// TIA Portal V15.1 export
// export: Created 2024-06-21T08:40:52.6402099Z, ExportSetting WithDefaults, DisplayName Totally Integrated Automation Portal, DisplayVersion V15.1 Update 5, DisplayName TIA Portal Openness, DisplayVersion V15.1 Update 5, DisplayName SINAMICS Startdrive Advanced, DisplayVersion V15.1, DisplayName G130, G150, S120, S150, SINAMICS MV, S210, DisplayVersion V15.1, DisplayName G110M, G120, G120C, G120D, G120P, DisplayVersion V15.1, DisplayName STEP 7 Professional, DisplayVersion V15.1 Update 5, DisplayName STEP 7 Safety, DisplayVersion V15.1, DisplayName WinCC Professional, DisplayVersion V15.1 Update 5, DisplayName SIMATIC Visualization Architect, DisplayVersion V15.1
FUNCTION_BLOCK "LHMIResetStart"   // FB1006, FBD
TITLE = LHMIResetStart
{ S7_Optimized_Access := 'FALSE' }
AUTHOR : VCC
FAMILY : Control
NAME : ModeSel
VERSION : 1.0
// ================================================================================
// This module is creating the needed integers for the F_ACK_OP module from reset 
// and start selections made on the HMI.  It also foresees the outputs for reset 
// and start to be connected to the modeselector.
// ================================================================================
// stored: AutoNumber false, IsIECCheckEnabled false, SetENOAutomatically False, UDAEnableTagReadback false
   VAR_INPUT
      I_SafetyNotOk { ExternalAccessible := 'False'; ExternalVisible := 'False'; ExternalWritable := 'False'} : Bool;   // Safety is not ok
      I_FailSafeResetAck { ExternalAccessible := 'False'; ExternalVisible := 'False'; ExternalWritable := 'False'} : Bool;   // F_Ack_Op FB in safety program is requesting value 9 on FailSafeReset output
      I_FailSafeAckID { ExternalAccessible := 'False'; ExternalVisible := 'False'; ExternalWritable := 'False'} : Int;   // F_Ack ID
   END_VAR
   VAR_OUTPUT
      O_HMIAlarmResetPBSel { ExternalAccessible := 'False'; ExternalVisible := 'False'; ExternalWritable := 'False'} : Bool;   // Alarm reset is activated
      O_HMIStartPBSel { ExternalAccessible := 'False'; ExternalVisible := 'False'; ExternalWritable := 'False'} : Bool;   // Start is activated
   END_VAR
   VAR_IN_OUT
      H_HMI1ModeCmd { ExternalAccessible := 'False'; ExternalVisible := 'False'; ExternalWritable := 'False'} : Word;   // Mode commands from HMI1
      IO_FailsafeReset { ExternalAccessible := 'False'; ExternalVisible := 'False'; ExternalWritable := 'False'} : Int;   // Number to Failsafe to reset safety
   END_VAR
   VAR DB_SPECIFIC
      HMI1Start { ExternalAccessible := 'False'; ExternalVisible := 'False'; ExternalWritable := 'False'} : Bool;   // Start on HMI1
      HMI1AlarmReset { ExternalAccessible := 'False'; ExternalVisible := 'False'; ExternalWritable := 'False'} : Bool;   // AlarmReset on HMI1
      HMI1AlarmResetAck { ExternalAccessible := 'False'; ExternalVisible := 'False'; ExternalWritable := 'False'} : Bool;   // Alarm Reset acknowledge from HMI1
      HMIAlarmResetPBSel { ExternalAccessible := 'False'; ExternalVisible := 'False'; ExternalWritable := 'False'} : Bool;   // Alarm reset is activated
      HMIStartPE { ExternalAccessible := 'False'; ExternalVisible := 'False'; ExternalWritable := 'False'} : Bool;   // Positive edge on start button from HMI
      HMIAlarmResetAckPE { ExternalAccessible := 'False'; ExternalVisible := 'False'; ExternalWritable := 'False'} : Bool;   // Positive edge on AlarmResetAck button from HMI
      AlarmResetPBSelReset { ExternalAccessible := 'False'; ExternalVisible := 'False'; ExternalWritable := 'False'} : Bool;   // Reset AlarmResetPBSel after predefined time
      AlarmResetPBSelResetPE { ExternalAccessible := 'False'; ExternalVisible := 'False'; ExternalWritable := 'False'} : Bool;   // Positive edge of AlarmResetPbSelReset
      FailSafeReset6Pulse { ExternalAccessible := 'False'; ExternalVisible := 'False'; ExternalWritable := 'False'} : Bool;   // Pulse to set value 6 on FailSafeReset Output
      FailSafeReset9Pulse { ExternalAccessible := 'False'; ExternalVisible := 'False'; ExternalWritable := 'False'} : Bool;   // Pulse to set value 9 on FailSafeReset Output
      ResetAlarmAckMemPulse { ExternalAccessible := 'False'; ExternalVisible := 'False'; ExternalWritable := 'False'} : Bool;   // Pulse to reset AlarmResetAckMem on negative edge of I_FailSafeResetAck
      AlarmResetAckMem { ExternalAccessible := 'False'; ExternalVisible := 'False'; ExternalWritable := 'False'} : Bool;   // memory : Pushbutton AlarmResetAck has been pushed on HMI
      FailsafeReset { ExternalAccessible := 'False'; ExternalVisible := 'False'; ExternalWritable := 'False'} : Int;   // Number to Failsafe to reset safety
   END_VAR
   VAR
      TimerAlarmResetPB { ExternalAccessible := 'False'; ExternalVisible := 'False'; ExternalWritable := 'False'} : "LTimer";
   END_VAR
   VAR_TEMP   // added for the SCL form of the ladder/FBD networks
      _w1 : Bool;
      _w2 : Bool;
   END_VAR
BEGIN

REGION Network 1: **** 1 - Inputs **** Extract the modeselection from HMI 1
   // Extract the modeselection from HMI 1
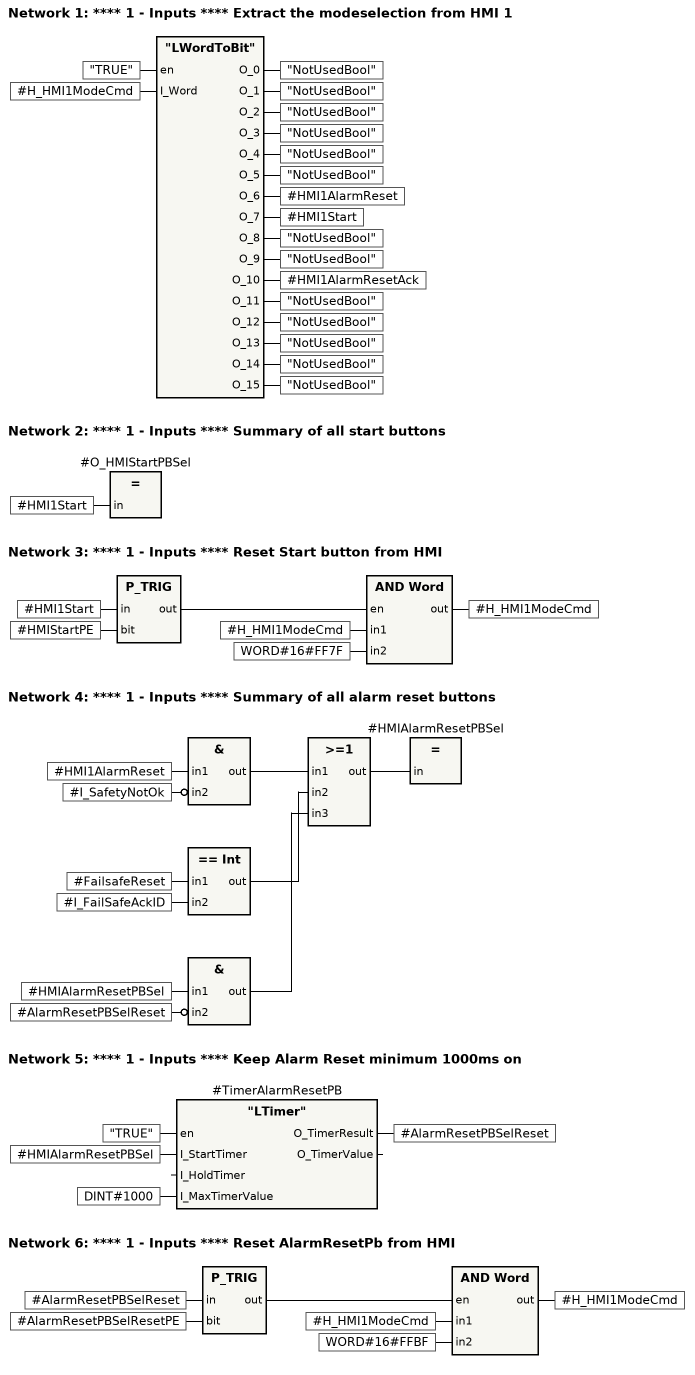
   IF "TRUE" THEN
       "LWordToBit"(I_Word := #H_HMI1ModeCmd,
                    O_0 => "NotUsedBool",
                    O_1 => "NotUsedBool",
                    O_2 => "NotUsedBool",
                    O_3 => "NotUsedBool",
                    O_4 => "NotUsedBool",
                    O_5 => "NotUsedBool",
                    O_6 => #HMI1AlarmReset,
                    O_7 => #HMI1Start,
                    O_8 => "NotUsedBool",
                    O_9 => "NotUsedBool",
                    O_10 => #HMI1AlarmResetAck,
                    O_11 => "NotUsedBool",
                    O_12 => "NotUsedBool",
                    O_13 => "NotUsedBool",
                    O_14 => "NotUsedBool",
                    O_15 => "NotUsedBool");
   END_IF;
END_REGION

REGION Network 2: **** 1 - Inputs **** Summary of all start buttons
   // Summary of all start buttons
   #O_HMIStartPBSel := #HMI1Start;
END_REGION

REGION Network 3: **** 1 - Inputs **** Reset Start button from HMI
   // Reset Start button from HMI
   #_w1 := #HMI1Start AND NOT #HMIStartPE;   // rising edge
   #HMIStartPE := #HMI1Start;
   IF #_w1 THEN #H_HMI1ModeCmd := #H_HMI1ModeCmd AND WORD#16#FF7F; END_IF;
END_REGION

REGION Network 4: **** 1 - Inputs **** Summary of all alarm reset buttons
   // Summary of all alarm reset buttons
   #HMIAlarmResetPBSel := (#HMI1AlarmReset AND NOT #I_SafetyNotOk) OR (#FailsafeReset = #I_FailSafeAckID) OR (#HMIAlarmResetPBSel AND NOT #AlarmResetPBSelReset);
END_REGION

REGION Network 5: **** 1 - Inputs **** Keep Alarm Reset minimum 1000ms on
   // Keep Alarm Reset minimum 1000ms on
   IF "TRUE" THEN
       #TimerAlarmResetPB(I_StartTimer := #HMIAlarmResetPBSel,   // "LTimer"
                          I_MaxTimerValue := DINT#1000,
                          O_TimerResult => #AlarmResetPBSelReset);
   END_IF;
END_REGION

REGION Network 6: **** 1 - Inputs **** Reset AlarmResetPb from HMI
   // Reset AlarmResetPb from HMI
   #_w1 := #AlarmResetPBSelReset AND NOT #AlarmResetPBSelResetPE;   // rising edge
   #AlarmResetPBSelResetPE := #AlarmResetPBSelReset;
   IF #_w1 THEN #H_HMI1ModeCmd := #H_HMI1ModeCmd AND WORD#16#FFBF; END_IF;
END_REGION

REGION Network 7: **** 1 - Inputs **** Reset AlarmResetAckPb from HMI
   // Reset AlarmResetAckPb from HMI
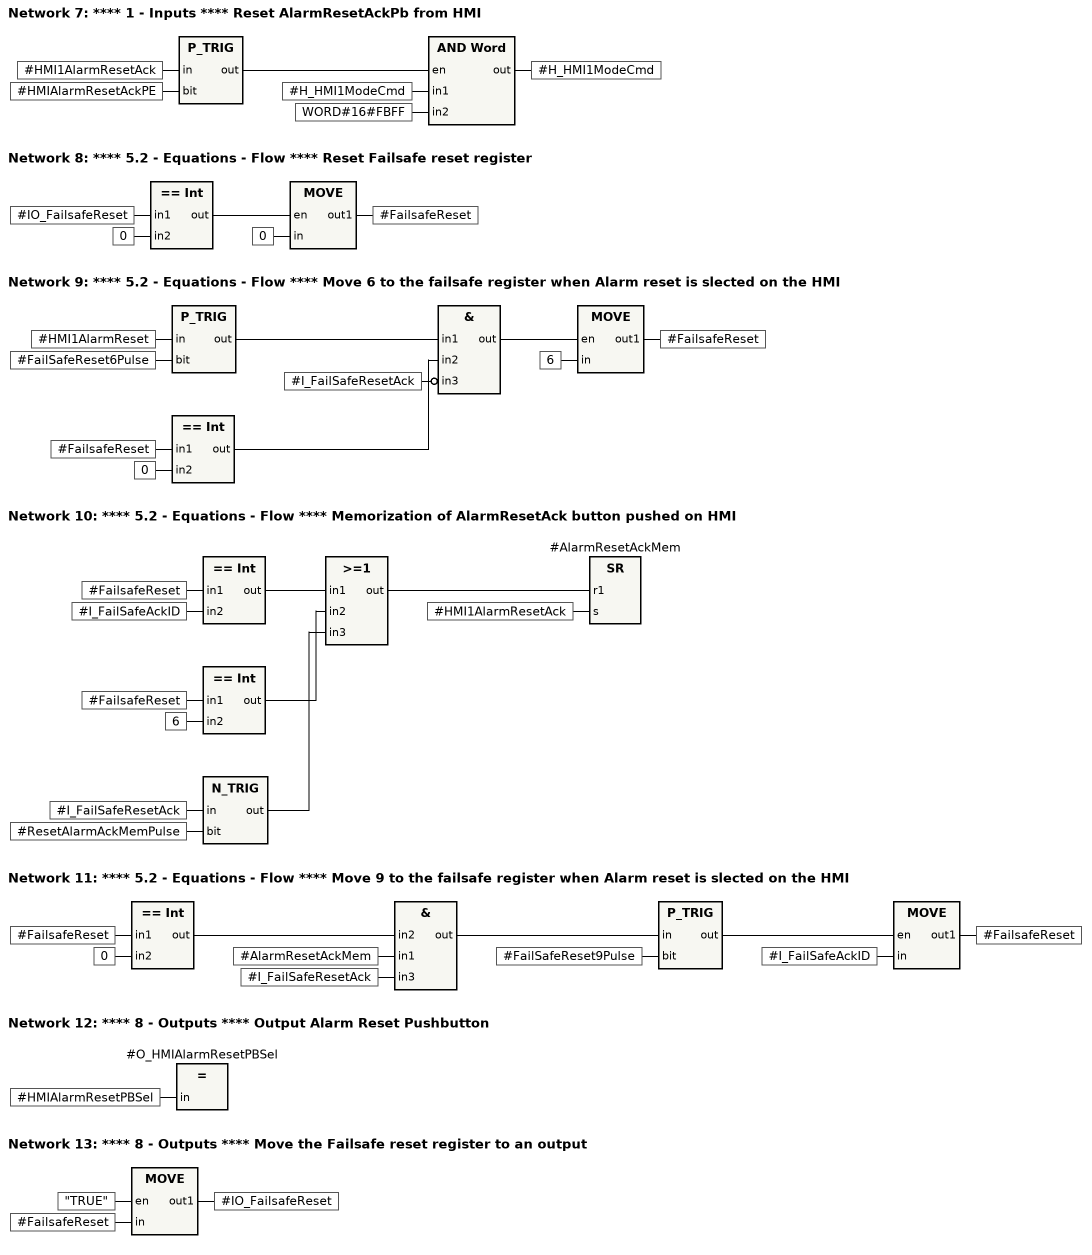
   #_w1 := #HMI1AlarmResetAck AND NOT #HMIAlarmResetAckPE;   // rising edge
   #HMIAlarmResetAckPE := #HMI1AlarmResetAck;
   IF #_w1 THEN #H_HMI1ModeCmd := #H_HMI1ModeCmd AND WORD#16#FBFF; END_IF;
END_REGION

REGION Network 8: **** 5.2 - Equations - Flow **** Reset Failsafe reset register
   // Reset Failsafe reset register
   IF #IO_FailsafeReset = 0 THEN #FailsafeReset := 0; END_IF;
END_REGION

REGION Network 9: **** 5.2 - Equations - Flow **** Move 6 to the failsafe register when Alarm reset is slected on the HMI
   // Move 6 to the failsafe register when Alarm reset is slected on the HMI
   #_w1 := #HMI1AlarmReset AND NOT #FailSafeReset6Pulse;   // rising edge
   #FailSafeReset6Pulse := #HMI1AlarmReset;
   IF #_w1 AND (#FailsafeReset = 0) AND NOT #I_FailSafeResetAck THEN #FailsafeReset := 6; END_IF;
END_REGION

REGION Network 10: **** 5.2 - Equations - Flow **** Memorization of AlarmResetAck button pushed on HMI
   // Memorization of AlarmResetAck button pushed on HMI
   #_w1 := NOT #I_FailSafeResetAck AND #ResetAlarmAckMemPulse;   // falling edge
   #ResetAlarmAckMemPulse := #I_FailSafeResetAck;
   IF #HMI1AlarmResetAck THEN
       #AlarmResetAckMem := TRUE;   // SR flip-flop
   END_IF;
   IF (#FailsafeReset = #I_FailSafeAckID) OR (#FailsafeReset = 6) OR #_w1 THEN
       #AlarmResetAckMem := FALSE;
   END_IF;
END_REGION

REGION Network 11: **** 5.2 - Equations - Flow **** Move 9 to the failsafe register when Alarm reset is slected on the HMI
   // Move 9 to the failsafe register when Alarm reset is slected on the HMI
   #_w1 := (#FailsafeReset = 0) AND #AlarmResetAckMem AND #I_FailSafeResetAck;
   #_w2 := #_w1 AND NOT #FailSafeReset9Pulse;   // rising edge
   #FailSafeReset9Pulse := #_w1;
   IF #_w2 THEN #FailsafeReset := #I_FailSafeAckID; END_IF;
END_REGION

REGION Network 12: **** 8 - Outputs **** Output Alarm Reset Pushbutton
   // Output Alarm Reset Pushbutton
   #O_HMIAlarmResetPBSel := #HMIAlarmResetPBSel;
END_REGION

REGION Network 13: **** 8 - Outputs **** Move the Failsafe reset register to an output
   // Move the Failsafe reset register to an output
   IF "TRUE" THEN #IO_FailsafeReset := #FailsafeReset; END_IF;
END_REGION
END_FUNCTION_BLOCK
